FUNCTION_BLOCK Valve_2DO
VAR_INPUT
	iOpen : BOOL;
	iClose : BOOL;
	iError : BOOL;
	iSecImp : BOOL;
END_VAR
VAR_OUTPUT
	oOpen : BOOL;
	oClose : BOOL;
END_VAR

VAR_IN_OUT
	ioValStruct	 : TValve;
END_VAR

VAR
	tempOpenStartupFail : BOOL;
	tempCloseStartupFail: BOOL;
END_VAR

{region "OpenState"}
    // set real state of valve input into valve structure - input of valve can be taken from limit sensor...
    ioValStruct.State.Open := iOpen;
    ioValStruct.State.Closed := iClose;
{endregion}

	 
{region "Manual/Automat"}
	// switching state of engine - automatic or manual control (default state is manual)
		 IF ioValStruct.Cmd.ManCtrl THEN
			ioValStruct.State.ManCtrl := TRUE;
			ioValStruct.State.AutCtrl :=FALSE;				 					  
		 END_IF
			  
		 IF ioValStruct.State.GenErr THEN
			ioValStruct.State.ManCtrl := TRUE;
			ioValStruct.State.AutCtrl :=FALSE;
		 END_IF
				 
	
		 IF ioValStruct.Cmd.AutCtrl THEN
			ioValStruct.State.ManCtrl := FALSE;
		    ioValStruct.State.AutCtrl := TRUE;					   
		 END_IF
			  
		IF (ioValStruct.Cmd.ManCtrl AND ioValStruct.Cmd.AutCtrl)	THEN
			ioValStruct.State.ManCtrl	:= TRUE;
			ioValStruct.State.AutCtrl	:= FALSE; 
		END_IF

    ioValStruct.Cmd.ManCtrl := FALSE;
    ioValStruct.Cmd.AutCtrl := FALSE;	
	
{endregion}
	
{region "MayRun / MayAutoRun"}
    // setting auxilary signals (may run, may auto run) - MR AND NOT MAR - engine may be started in manual mode, MAR - engine may be started in automatic mode
    ioValStruct.State.MayRun := (ioValStruct.State.ManCtrl AND NOT(ioValStruct.State.GenErr));
	ioValStruct.State.MayAutoRun := (ioValStruct.State.AutCtrl AND NOT(ioValStruct.State.GenErr));
{endregion}
	 
{region "ManCtrl"}
	// processing manual actions - if command is processed, it is sets to FALSE even if can't be processed
    // Valve commands are open, close and stop - valve can be stopped intermediate position
	 IF ioValStruct.State.ManCtrl AND ioValStruct.State.MayRun THEN
        IF ioValStruct.Cmd.OpenMan THEN
            ioValStruct.State.CloseOut := FALSE;
            ioValStruct.State.OpenOut := TRUE;
        END_IF;
        
        IF ioValStruct.Cmd.CloseMan THEN
            ioValStruct.State.OpenOut := FALSE;
            ioValStruct.State.CloseOut := TRUE;
        END_IF;
        
        IF ioValStruct.Cmd.StopMan THEN
            ioValStruct.State.OpenOut := FALSE;
            ioValStruct.State.CloseOut := TRUE;
        END_IF;
    END_IF;
    
    ioValStruct.Cmd.OpenMan := FALSE;
    ioValStruct.Cmd.CloseMan := FALSE;
    ioValStruct.Cmd.StopMan := FALSE;
{endregion}
	 
{region "AutCtrl"}
	 //if request to run in automatic mode -> set outputs to right states if MAR
    //AutoRequest shouldn't be reseted to false state
    //if request to open and request to close are setted to 1 simultaneously - outputs should be 0.
    IF ioValStruct.State.AutCtrl AND ioValStruct.State.MayAutoRun THEN
        IF ioValStruct.Cmd.Req2CloseAut AND (NOT ioValStruct.Cmd.Req2OpenAut) THEN
            ioValStruct.State.OpenOut := FALSE;
            ioValStruct.State.CloseOut := TRUE;
        END_IF;
        
        IF (NOT ioValStruct.Cmd.Req2CloseAut) AND ioValStruct.Cmd.Req2OpenAut THEN
            ioValStruct.State.CloseOut := FALSE;
            ioValStruct.State.OpenOut := TRUE;
        END_IF;
        
        IF (NOT ioValStruct.Cmd.Req2CloseAut) AND (NOT ioValStruct.Cmd.Req2OpenAut) THEN
            ioValStruct.State.CloseOut := FALSE;
            ioValStruct.State.OpenOut := FALSE;
        END_IF;
        
    END_IF;
{endregion}
	 
{region "Error states"}
 // definition of error states 
    // error - input from digital input of plc - fyzical state of valve
    // calculating start up fail - if output is sets to open or close, it's expected feedback from limit sensor in defined time, if feedback doesn't show in this time, it should be start up fail error
    // merge of these two error is general error
    // error is both inputs (open and closed) true state
    ioValStruct.OpenFailTimer(IN := (ioValStruct.State.OpenOut AND (NOT ioValStruct.State.CloseOut)), PT := ioValStruct.Time2Open);
	IF	ioValStruct.OpenFailTimer.Q AND NOT ioValStruct.State.Open	THEN	//MANDATORY CONDITION (I had to add Input from sensor)
		tempOpenStartupFail := TRUE;								
	END_IF

    ioValStruct.CloseFailTimer(IN := ((NOT ioValStruct.State.OpenOut) AND ioValStruct.State.CloseOut), PT := ioValStruct.Time2Open);
	IF	ioValStruct.OpenFailTimer.Q AND NOT ioValStruct.State.Open	THEN	//MANDATORY CONDITION (I had to add Input from sensor)
		tempCloseStartupFail := TRUE;							
	END_IF	

    
   
    IF tempOpenStartupFail OR tempCloseStartupFail THEN
        ioValStruct.State.StartUpFail := TRUE;
    END_IF;
    
    IF iError THEN
        ioValStruct.State.Err := TRUE;
    END_IF;
    
    ioValStruct.State.GenErr := ioValStruct.State.StartUpFail OR iError;
    
    // start up fail can be reseted by operator, command resetSUF, resets SUF and engine should be started again
    IF ioValStruct.Cmd.ResetSUF THEN
        ioValStruct.State.StartUpFail := FALSE;
        ioValStruct.Cmd.ResetSUF := FALSE;
    END_IF;
    
    // if error state exists outputs should be in stop state
    IF ioValStruct.State.GenErr THEN
        ioValStruct.State.OpenOut := FALSE;
        ioValStruct.State.CloseOut := FALSE;
    END_IF;
{endregion}
	 	 
oOpen := ioValStruct.State.OpenOut;
oClose := ioValStruct.State.CloseOut;

{region "StatusInt"}
    //write combination of states into int value for visualization (valve - combination of open, close state and error)
    IF ioValStruct.State.Open AND NOT ioValStruct.State.Closed AND NOT ioValStruct.State.GenErr THEN
        ioValStruct.State.StColor := Global.Open;
    ELSIF NOT ioValStruct.State.Open AND ioValStruct.State.Closed AND NOT ioValStruct.State.GenErr THEN
        ioValStruct.State.StColor := Global.Closed;
    ELSIF ioValStruct.State.Open AND NOT ioValStruct.State.Closed AND ioValStruct.State.GenErr THEN
        ioValStruct.State.StColor := Global.OpenAndErr;
    ELSIF NOT ioValStruct.State.Open AND ioValStruct.State.Closed AND ioValStruct.State.GenErr THEN
        ioValStruct.State.StColor := Global.ClosedAndErr;
    ELSIF NOT ioValStruct.State.Open AND NOT ioValStruct.State.Closed AND NOT ioValStruct.State.GenErr THEN
        ioValStruct.State.StColor := Global.NotOpenNotClosedNotErr;
    ELSIF NOT ioValStruct.State.Open AND NOT ioValStruct.State.Closed AND ioValStruct.State.GenErr THEN
        ioValStruct.State.StColor := Global.NotOpenNotClosedAndErr;
    ELSIF ioValStruct.State.Open AND ioValStruct.State.Closed AND ioValStruct.State.GenErr THEN
        ioValStruct.State.StColor := Global.OpenAndClosedAndErr;
    ELSIF ioValStruct.State.Open AND ioValStruct.State.Closed AND NOT ioValStruct.State.GenErr THEN
        ioValStruct.State.StColor := Global.OpenAndClosedNotErr;
    END_IF;
{endregion}

END_FUNCTION_BLOCK

(* stored: Version 1.1.0.1, ProductVersion 3.1.4024.15
   POU Valve_2DO: Id {86469f36-9490-4936-ae7d-f4831ca2b758}, SpecialFunc None *)
